{attribute 'qualified_only'}
{attribute 'strict'}
{attribute 'to_string'}
TYPE E_EStop :
(
	Activated		:=0,
	Normallyclosed 	:=3

)BYTE;
END_TYPE

(* stored: Version 1.1.0.1, ProductVersion 3.1.4026.19
   DUT E_EStop: Id {43baa300-64bb-4889-99c6-d9f49fbabdcc} *)
